// TIA Portal V18 export
// export: Created 2026-03-12T15:56:19.279516Z, ExportSetting WithDefaults, DisplayName Totally Integrated Automation Portal, DisplayVersion V18 Update 5, DisplayName TIA Portal Openness, DisplayVersion V18 Update 5, DisplayName TIA Portal Version Control Interface, DisplayVersion V18, DisplayName SINAMICS Startdrive Advanced, DisplayVersion V18, DisplayName SINAMICS Startdrive G130, G150, S120, S150, SINAMICS MV, S210, DisplayVersion V18, DisplayName SINAMICS Startdrive G110M, G120, G120C, G120D, G120P, G115D, DisplayVersion V18, DisplayName STEP 7 Professional, DisplayVersion V18 Update 5, DisplayName STEP 7 Safety, DisplayVersion V18, DisplayName WinCC Professional, DisplayVersion V18 Update 5
DATA_BLOCK "FB SUCÇÃO OK BH-01A"   // DB214
VERSION : 0.1
// stored: AutoNumber true, DBAccessibleFromOPCUA true, DBAccessibleFromWebserver true, InstanceOfName FB SUCÇÃO OK, InstanceOfType FB
"FB SUCÇÃO OK"
   // VAR_INPUT
   //    REFERENCIA : Real;
   //    CADASTRO_SUCÇAO_INSUFICIENTE : Real;
   //    CADASTRO_TEMPO_RESET : Time;
   // END_VAR
   // VAR_OUTPUT
   //    SUCÇÃO_OK : Bool;
   // END_VAR
   // VAR
   //    SUCCAO_INSUFICIENTE : Bool;
   //    RESET_ALARME : IEC_TIMER;
   // END_VAR
BEGIN
END_DATA_BLOCK
